(* PLC project motor1dir_1speed, Dassault Systèmes ControlBuild 2024x Refresh1 *)
(* stored: creationDateTime 2024-01-23T16:33:10-01:00 *)

CONFIGURATION motor1dir_1speed
  VAR_GLOBAL
    simuperiod : REAL := 50000.0;
    taskname : STRING(50) := 'motor1dir_1speed.exe';
    allowpreconditions : BOOL := true;
    allowpostconditions : BOOL := true;
  END_VAR
END_CONFIGURATION
